PROGRAM MAIN
VAR
	// To controller
	fWRefPrep								: LREAL := 0;
	
	fThetaOl								: REAL := 0;
	
	// Encoder
	bHomingDoneEncoder						: BOOL;
	uEncoderOffset							: UINT;
	
	fCurrentMeasurement_V					: REAL; // Current measurement as voltage
	fCurrent_I								: REAL; // Current as A
	fMotorSpeed								: REAL;
	fThetaOut, fThetaElOut, fOmegaOut	 	: REAL;
	
	fTheta 									: REAL;
	fThetaEl 								: REAL;
	fOmega									: REAL;
	fVa, fVb								: REAL;
	
	bControlEnable							: BOOL := FALSE;
	bstartHoming							: BOOL := FALSE;
	bOpenLoop 								: BOOL := FALSE;
	bHomingDone 							: BOOL := FALSE;
	fHomingVa								: REAL := 0.5;
	fHomingVb								: REAL := 0;
	
	fbCAN_MessageHandler					: FB_CANMessageHandler();
	fbEncoder								: FB_Encoder();
	
	stInputs								: ST_Inputs;
	stOutputs								: ST_Outputs;
END_VAR


//control_enable := 0;
IF bControlEnable THEN
	stOutputs.fControlEnable := 1;
ELSE	
	stOutputs.fControlEnable := 0;
END_IF 

stOutputs.fWref := fWRefPrep * 2;

stOutputs.fIa := F_VoltageToCurrentConvert(F_AnalogIntToVoltage(stInputs.uEL3702Ch1_In));
stOutputs.fIb := F_VoltageToCurrentConvert(F_AnalogIntToVoltage(stInputs.uEL3702Ch2_In));
stOutputs.fIc := F_VoltageToCurrentConvert(F_AnalogIntToVoltage(stInputs.uEL3702Ch3_In));

//IF ( Measurements.COUNTER_VALUE > Constants.PULSES_PER_REV ) AND (EL5101_CounterSetWORD.2 = FALSE) THEN
//	EL5101_CounterSet := Constants.PULSES_PER_REV - (16#FFFF - Measurements.COUNTER_VALUE);
//	EL5101_CounterSetWORD.2 := TRUE;
//ELSE
//	EL5101_CounterSetWORD.2 := FALSE;
//END_IF

fbEncoder(	fThetaEl => stOutputs.fTcTheta,
			fThetaMech => stOutputs.fThetaMech,
			fOmegaEl => stOutputs.fWactual,
			fOmegaMech => stOutputs.fWmech);
			
fVa := LREAL_TO_REAL(stInputs.fAlpha_U);
fVb := LREAL_TO_REAL(stInputs.fBeta_U);

IF bStartHoming THEN
	stOutputs.fControlEnable := 0;
	//fbHomingTimer(DONE => homingDone);
	fbCAN_MessageHandler(Inputs := stInputs.Inputs, 
						Outputs := stOutputs.Outputs, 
						fVoltage_A := fHomingVa,
						fVoltage_B := fHomingVb);
	uEncoderOffset := stInputs.uEL5101_Counter;
	bHomingDone := TRUE;
END_IF

IF (NOT bStartHoming) AND bHomingDone THEN
	bHomingDoneEncoder := 1;
	
	IF bControlEnable THEN
		fbCAN_MessageHandler(Inputs := stInputs.Inputs, 
							Outputs := stOutputs.Outputs, 
							fVoltage_A := fVa,
							fVoltage_B := fVb);
	ELSIF bOpenLoop THEN
		fbCAN_MessageHandler(Inputs := stInputs.Inputs, 
							Outputs := stOutputs.Outputs, 
							fVoltage_A := SIN(fThetaOl),
							fVoltage_B := COS(fThetaOl));
		
		fThetaOl := fThetaOl + 2 * LREAL_TO_REAL( PI ) / 2500;
		IF fThetaOl > 2 * PI THEN
			fThetaOl := 0;
		END_IF
	END_IF
	
(*	
ELSE
	fbCAN_MessageHandler(	Inputs := Inputs, 
						Outputs := Outputs, 
						fVoltage_A := homingVa,
						fVoltage_B := homingVb);
	EL5101_CounterSet := 0;*)
END_IF

END_PROGRAM

(* stored: Version 1.1.0.1, ProductVersion 3.1.4024.11
   POU MAIN: Id {bdfa0062-539d-4679-9449-b5aad24542ad}, SpecialFunc None *)
